// TIA Portal V18 export
DATA_BLOCK "Pallets_Stations"   // DB11
{ S7_Optimized_Access := 'TRUE' }
// stored: MemoryReserve 100
   VAR
      Pallets : Array[1..24] of "Pallet";
      Stations : Array[1..4, 1..12] of "Station";
   END_VAR
BEGIN
END_DATA_BLOCK
